{attribute 'linkalways'}
{attribute 'no_explicit_call' := 'do not call this POU directly'}
FUNCTION_BLOCK InstanceRemovedEvent EXTENDS Event IMPLEMENTS I_InstanceRemovedEvent
VAR
	_instance : I_Instance;
END_VAR

PROPERTY PUBLIC Instance : I_Instance
GET
Instance := _instance;
END_GET
END_PROPERTY

METHOD PUBLIC Notify
VAR_INPUT
	Instance : I_Instance;
END_VAR
_instance := instance;
NotifySubscribers();
END_METHOD

END_FUNCTION_BLOCK

(* stored: Version 1.1.0.1, ProductVersion 3.1.4024.11
   POU InstanceRemovedEvent: Id {227f2fc3-0115-4986-9712-4ba0d0df4526}, SpecialFunc None
   Property Instance: Id {1f253a84-dc7a-4c27-8a4b-538ae767b11c}
   Get Get: Id {4e7b4e23-c9cc-444f-99ba-1b8dfbe37bfa}
   Method Notify: Id {3f18c54f-f9ce-4136-99a6-703b5bcb05cc} *)
